SUBAPPLICATION Softkey_Aux_Method_IE (* SoftKey ODER AUX (Joystick, via Softkey_Aux_IE) ODER lokale argumentlose OPC-UA-Methode (ACTION=CREATE_METHOD, SERVER_0 - z.B. von Web-Client/vt-ui-mirror oder OPC-Dashboard aufgerufen) aktiviert -> 1 gemeinsames IND-Event. Baut auf Softkey_Aux_IE auf und ergaenzt den Methoden-Kanal - Gegenstueck zu Softkey_Aux_Web_IE (dort: Web per SUBSCRIBE_R_TRIG auf eine geschriebene Variable, hier: Web/Dashboard per echtem RPC-Methodenaufruf, keine gemeinsame Variable). *)
  (* Standard: 61499-2; Description: Copyright (c) 2026 Meisterschulen am Ostbahnhof This program and the accompanying materials are made available under the terms of the Eclipse Public License 2.0 which is available at https://www.eclipse.org/legal/epl-2.0/ SPDX-License-Identifier: EPL-2.0 *)
  (* Version 1.0, 2026-09-11, Franz Höpfinger, Meisterschulen am Ostbahnhof, initial implementation - herausgeloest aus AX_SoftkeyToggle_RS_TO_QXA_BG (Softkey_Aux_IE + SERVER_0 kam dort 2x vor, fuer Toggle und fuer Reset), wiederverwendbar fuer jeden Event-Trigger, der per SoftKey/AUX/Web-Methode/Dashboard gleichberechtigt ausgeloest werden soll. *)
  PACKAGE MyLib::sys;
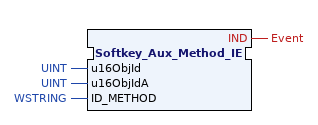
  EVENT_OUTPUT
    IND; (* Feuert wenn SoftKey, AUX ODER die lokale Methode aktiviert/aufgerufen wird *)
  END_EVENT
  VAR_INPUT
    u16ObjId : UINT; (* Object ID SoftKey *)
    u16ObjIdA : UINT; (* Object ID AuxFunction2 *)
    ID_METHOD : WSTRING; (* Lokale Methodenadresse (ACTION=CREATE_METHOD) fuer den argumentlosen Trigger - wird von Web-Client (vt-ui-mirror) UND direkt vom OPC-Dashboard aufgerufen *)
  END_VAR
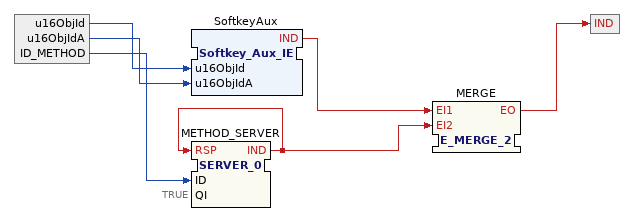
  (* RSP MUSS auf IND zurueckverdrahtet werden (argumentloser Trigger, keine Verarbeitung noetig) - sonst blockiert FORTEs onServerMethodCall den OPC-UA-Server-Thread bis zu 4s und haelt dabei open62541s globalen serviceMutex, den JEDER AX_PUBLISH_1 auf einem anderen FORTE-Thread ebenfalls braucht. Siehe Ventilsteuerung/OPC_UA_VERNETZUNG.md Punkt 12. *)
  FBS
    METHOD_SERVER : iec61499::net::SERVER_0(QI := TRUE);
    MERGE : iec61499::events::E_MERGE_2;
  END_FBS
  SUBAPPS
    SoftkeyAux : MyLib::sys::Softkey_Aux_IE;
  END_SUBAPPS
  EVENT_CONNECTIONS
    SoftkeyAux.IND TO MERGE.EI1;
    METHOD_SERVER.IND TO MERGE.EI2;
    METHOD_SERVER.IND TO METHOD_SERVER.RSP;
    MERGE.EO TO IND;
  END_CONNECTIONS
  DATA_CONNECTIONS
    u16ObjId TO SoftkeyAux.u16ObjId;
    u16ObjIdA TO SoftkeyAux.u16ObjIdA;
    ID_METHOD TO METHOD_SERVER.ID;
  END_CONNECTIONS
END_SUBAPPLICATION
